// TwinCAT 3 PLC project Untitled1
// ProgramVersion: 3.1.4023.0
// libraries:
//   CmpBitmapPool, * (System)
//   Tc2_Standard, * (Beckhoff Automation GmbH)
//   Tc2_System, * (Beckhoff Automation GmbH)
//   Tc2_Utilities, * (Beckhoff Automation GmbH)
//   Tc3_Module, * (Beckhoff Automation GmbH)
// project tree:
//   / GlobalTextList.TcGTLO, PlcTask.TcTTO, Visualization Manager.TcVMO (not stored)
//   POUs/ MAIN.TcPOU
//   VISUs/ ImagePool.TcIPO (not stored), TextList.TcTLO, Visualization_1.TcVIS, Visualization_2.TcVIS, Visualization_3.TcVIS, VISU_FRAME.TcVIS
// real-time tasks:
//   TASK PlcTask: cycle T#10ms, priority 20, ADS port 350

CONFIGURATION Untitled1
    RESOURCE PLC ON TwinCAT3
        TASK PlcTask(INTERVAL := T#10ms, PRIORITY := 20);
        PROGRAM MAIN WITH PlcTask : MAIN;
    END_RESOURCE
END_CONFIGURATION

// ---- POUs/MAIN.TcPOU
PROGRAM MAIN
VAR
	nState: INT;
	bButton: BOOL;
	ftrig1: F_TRIG;
	bSensor1: BOOL;
	bHat: BOOL;
	rtrig1: R_TRIG;
	bSensor2: BOOL;
	Random1: DRAND;
	nYukseklik: INT;
	sMsgInfo: STRING;
	T1: TON;
	bValf1: BOOL;
	rtrig_Kutu1: R_TRIG;
	rtrig_Kutu2: R_TRIG;
	rtrig_Kutu3: R_TRIG;
	bKutuSensor_1: BOOL;
	bKutuSensor_2: BOOL;
	bKutuSensor_3: BOOL;
	nMalzeme1: INT;
	bValf2: BOOL;
	nMalzeme2: INT;
	bValf3: BOOL;
	nMalzeme3: INT;
	sMsgKisa: STRING(255);
	sMsgOrta: STRING(255);
	sMsgUzun: STRING(255);
	sMsgMalzemeInfo: STRING(255);
	fbSystemTime: FB_LocalSystemTime;
	Year: STRING;
	Month: STRING;
	Day: STRING;
	DMY_LocalTime: STRING;
	HMS_LocalTime: STRING(255);
	Sec: STRING(255);
	Hours: STRING;
	Minute: STRING;
END_VAR



ACT_Uygulama1();
ACT_VisuString();

ACTION ACT_Uygulama1:


ftrig1(CLK:= bSensor1 , Q=> ); // Hattın başında malzeme var mı ?
rtrig1(CLK:= bSensor2 , Q=> ); // Ölçüm yapılacak yerde malzeme var mı ?

rtrig_Kutu1(CLK:= bKutuSensor_1 , Q=> );	// Kısa Boyutlu Malzeme düştü mü kontrolü 
rtrig_Kutu2(CLK:= bKutuSensor_2 , Q=> );	// Orta Boyutlu Malzeme düştü mü kontrolü 
rtrig_Kutu3(CLK:= bKutuSensor_3 , Q=> );	// Uzun Boyutlu Malzeme düştü mü kontrolü 

CASE nState OF
	
	0:
	
		IF bButton THEN 
			
			nState := 10;
			
		END_IF
		
	10:
	
	sMsgInfo := 'Yeni Malzemenin Hatta Aktarılması Bekleniyor';
	
		IF ftrig1.Q THEN
			
			bHat := TRUE;			
			nState := 20;
			
		END_IF
		
	20:
	
	sMsgInfo := 'Malzemenin İstenilen Konuma Gelmesi Bekleniyor';
	
		IF rtrig1.Q THEN
			
			bHat := FALSE;
			
			Random1(Seed:=0 , Num=> );			
			nYukseklik := LREAL_TO_INT((Random1.Num)*100);
			
			nState := 30;
			
		END_IF
	
	30:
	
		IF nYukseklik >= 0 AND nYukseklik <= 30 THEN
			
			nState := 32;
			sMsgInfo := 'Kısa Boyutlu Malzeme.';
		
		ELSIF nYukseklik >30 AND nYukseklik <= 65 THEN

			nState := 34;
			sMsgInfo := 'Orta Boyutlu Malzeme.';

		ELSIF nYukseklik >65 AND nYukseklik <= 100 THEN

			nState := 36;
			sMsgInfo := 'Uzun Boyutlu Malzeme.';
		ELSE 
			sMsgInfo := 'HATA...!';
			nState := 999;
			
		END_IF
		
	32:
	
		bHat := TRUE;
		T1(IN:=TRUE , PT:= T#2S);
		
		IF T1.Q THEN
			nState := 42;
			T1(IN := FALSE);
			bHat := FALSE;
		END_IF
	
	34:
	
		bHat := TRUE;
		T1(IN:=TRUE , PT:= T#4S);
		
		IF T1.Q THEN
			nState := 44;
			T1(IN := FALSE);
			bHat := FALSE;
		END_IF
	
	36:
	
		bHat := TRUE;
		T1(IN:=TRUE , PT:= T#6S);
		
		IF T1.Q THEN
			nState := 46;
			T1(IN := FALSE);
			bHat := FALSE;
		END_IF
		
	42:
	
		bValf1 := TRUE;
		
		sMsgInfo := 'Kısa Boyutlu Malzeme Kutusuna Aktarılıyor.';
		
		IF rtrig_Kutu1.Q THEN
			
			bValf1 := FALSE;
			
			nMalzeme1 := nMalzeme1 + 1; // Kısa boyutlu malzeme sayısını 1 arttır.
			
			nState := 0;
			
		END_IF
		
		
	
	44:
		bValf2 := TRUE;
		
		sMsgInfo := 'Orta Boyutlu Malzeme Kutusuna Aktarılıyor.';
		
		IF rtrig_Kutu2.Q THEN
			
			bValf2 := FALSE;
			
			nMalzeme2 := nMalzeme2 + 1; // Kısa boyutlu malzeme sayısını 1 arttır.
			
			nState := 0;
			
		END_IF
	
	46:
	
		bValf3 := TRUE;
		
		sMsgInfo := 'Uzun Boyutlu Malzeme Kutusuna Aktarılıyor.';
		
		IF rtrig_Kutu3.Q THEN
			
			bValf3 := FALSE;
			
			nMalzeme3 := nMalzeme3 + 1; // Kısa boyutlu malzeme sayısını 1 arttır.
			
			nState := 0;
			
		END_IF
	
		
		
END_CASE

IF NOT bButton THEN
	
	sMsgInfo := 'Sistem Kapalı Durumda.';
	
	nState := 0;
	
	bValf1 := FALSE;
	bValf2 := FALSE;
	bValf3 := FALSE;
	
	bHat := FALSE;
	
	T1(IN:=FALSE);
	
END_IF
END_ACTION

ACTION ACT_VisuString:



sMsgKisa := CONCAT(STR1:='Kısa Boyutlu Malzeme Kutusunda ' , STR2:=INT_TO_STRING(nMalzeme1));
sMsgKisa := CONCAT(STR1:=sMsgKisa , STR2:=' Malzeme Var.' );

sMsgOrta := CONCAT(STR1:='Orta Boyutlu Malzeme Kutusunda ' , STR2:=INT_TO_STRING(nMalzeme2));
sMsgOrta:= CONCAT(STR1:=sMsgOrta , STR2:=' Malzeme Var.' );

sMsgUzun := CONCAT(STR1:='Uzun Boyutlu Malzeme Kutusunda ' , STR2:=INT_TO_STRING(nMalzeme3));
sMsgUzun := CONCAT(STR1:=sMsgUzun , STR2:=' Malzeme Var.' );

sMsgMalzemeInfo := CONCAT(STR1:='Malzeme Boyutu: ' , STR2:=INT_TO_STRING(nYukseklik));
sMsgMalzemeInfo := CONCAT(STR1:=sMsgMalzemeInfo , STR2:='[cm]' );



fbSystemTime(	bEnable:=TRUE );


Year 	:= 	WORD_TO_STRING(fbSystemTime.systemTime.wYear);
Month	:= 	WORD_TO_STRING(fbSystemTime.systemTime.wMonth);
Day 	:= 	WORD_TO_STRING(fbSystemTime.systemTime.wDay);

Hours	:=	WORD_TO_STRING(	fbSystemTime.systemTime.wHour);
Minute	:=  WORD_TO_STRING( fbSystemTime.systemTime.wMinute);
Sec		:=	WORD_TO_STRING( fbSystemTime.systemTime.wSecond);


DMY_LocalTime := CONCAT(STR1:=Day , STR2:='/' );
DMY_LocalTime := CONCAT(STR1:=DMY_LocalTime , STR2:= Month);
DMY_LocalTime := CONCAT(STR1:=DMY_LocalTime , STR2:='/' );
DMY_LocalTime := CONCAT(STR1:=DMY_LocalTime , STR2:=Year );


HMS_LocalTime	:=	CONCAT(STR1:=Hours , STR2:=':' );	
HMS_LocalTime	:=	CONCAT(STR1:=HMS_LocalTime , STR2:=Minute );
HMS_LocalTime	:=	CONCAT(STR1:=HMS_LocalTime , STR2:=':' );	
HMS_LocalTime	:=	CONCAT(STR1:=HMS_LocalTime , STR2:=Sec );
END_ACTION

END_PROGRAM

// ---- GlobalTextList.TcGTLO
TEXTLIST GlobalTextList
  624 = '%s'
  684 = 'Ana Ekran'
  849 = 'Ana Sayfa'
  63 = 'bSensor1'
  479 = 'bSensor2'
  706 = 'Dil Seçeneği'
  637 = 'GroupBox'
  441 = 'Konveyör Hattı'
  907 = 'KutuSensor1'
  970 = 'KutuSensor2'
  179 = 'KutuSensor3'
  389 = 'Sensor Kontrol Bölümü'
  742 = 'Sensor1'
  268 = 'Sensor2'
  823 = 'Sensörler'
  410 = 'Sistem'
  646 = 'Sistem Kontrol'
  207 = 'Türkçe'
  940 = 'Valf1'
  808 = 'Valf2'
  708 = 'Valf3'
  488 = 'Çıkışlar'
  996 = 'İngilizce'
END_TEXTLIST

// ---- VISUs/TextList.TcTLO
TEXTLIST TextList
  0 = 'Sistem' | Türkçe: 'Sistem' | İngilizce: 'System'
  1 = 'Dil Seçeneği' | Türkçe: 'Dil Seçeneği' | İngilizce: 'Languages'
  2 = 'Ana Sayfa' | Türkçe: 'Ana Sayfa' | İngilizce: 'Home Page'
  3 = 'İngilizce' | Türkçe: 'İngilizce' | İngilizce: 'English'
  4 = 'Türkçe' | Türkçe: 'Türkçe' | İngilizce: 'Turkish'
   = ''
END_TEXTLIST

// ---- VISUs/Visualization_1.TcVIS
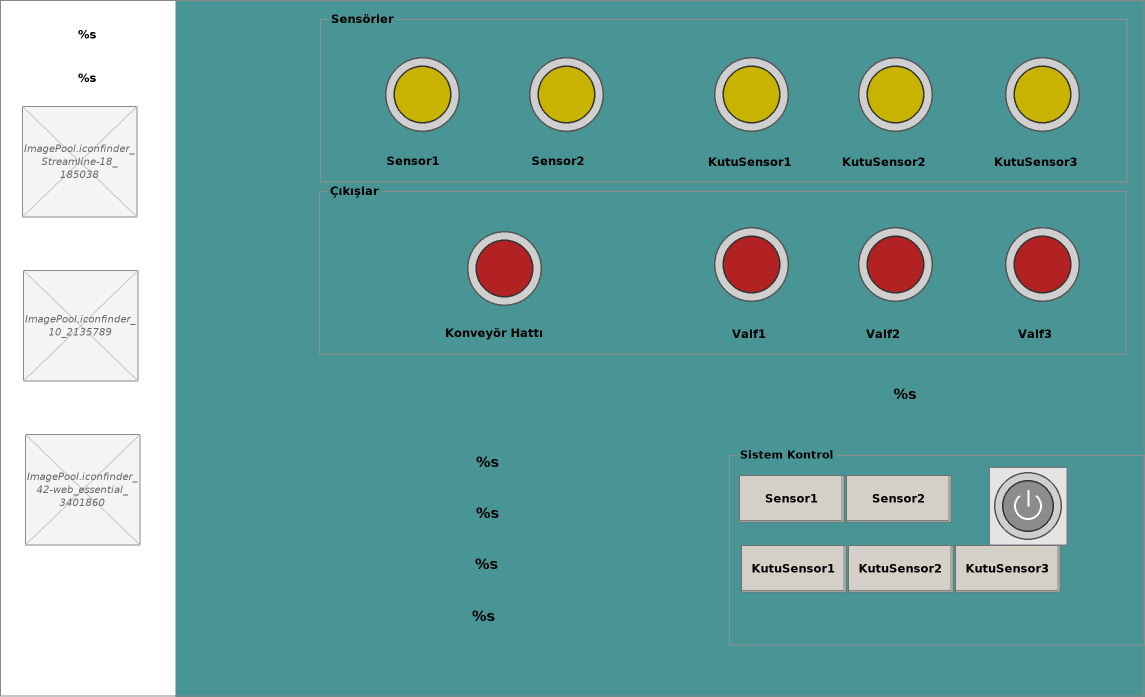
VISUALIZATION Visualization_1  // 1145x697
    Button (739,475 105x47), "Sensor1"
        toggle MAIN.bSensor1
    Button (846,475 105x47), "Sensor2"
        toggle MAIN.bSensor2
    Button (741,545 105x47), "KutuSensor1"
        toggle MAIN.bKutuSensor_1
    Button (848,545 105x47), "KutuSensor2"
        toggle MAIN.bKutuSensor_2
    Button (955,545 105x47), "KutuSensor3"
        toggle MAIN.bKutuSensor_3
    Lamp1 (370,51 105x87), variable: MAIN.bSensor1, style: Lamp-Lamp1-Yellow
    Lamp1 (514,51 105x87), variable: MAIN.bSensor2, style: Lamp-Lamp1-Yellow
    Lamp1 (699,51 105x87), variable: MAIN.bKutuSensor_1, style: Lamp-Lamp1-Yellow
    Lamp1 (843,51 105x87), variable: MAIN.bKutuSensor_2, style: Lamp-Lamp1-Yellow
    Lamp1 (990,51 105x87), variable: MAIN.bKutuSensor_3, style: Lamp-Lamp1-Yellow
    GroupBox (320,11 807x171), "Sensörler"
        Label (42,135 102x30), "Sensor1"
        Label (187,135 102x30), "Sensor2"
        Label (379,136 102x30), "KutuSensor1"
        Label (513,136 102x30), "KutuSensor2"
        Label (665,136 102x30), "KutuSensor3"
    Lamp1 (699,221 105x87), variable: MAIN.bValf1, style: Lamp-Lamp1-Red
    Lamp1 (843,221 105x87), variable: MAIN.bValf2, style: Lamp-Lamp1-Red
    Lamp1 (990,221 105x87), variable: MAIN.bValf3, style: Lamp-Lamp1-Red
    GroupBox (319,183 807x171), "Çıkışlar"
        Label (124,135 102x30), "Konveyör Hattı"
        Label (379,136 102x30), "Valf1"
        Label (513,136 102x30), "Valf2"
        Label (665,136 102x30), "Valf3"
        Lamp1 (133,42 105x87), variable: MAIN.bHat, style: Lamp-Lamp1-Red
    Rectangle (271,440 433x44), "%s", text variable: MAIN.sMsgInfo, text list: ''
    Rectangle (270,491 435x44), "%s", text variable: MAIN.sMsgKisa
    Rectangle (267,542 439x44), "%s", text variable: MAIN.sMsgOrta
    Rectangle (259,594 449x44), "%s", text variable: MAIN.sMsgUzun
    Rectangle (746,372 318x44), "%s", text variable: MAIN.sMsgMalzemeInfo
    Frame (0,0 175x697)
        shows VISU_FRAME(sDayTime := MAIN.DMY_LocalTime, sTime := MAIN.HMS_LocalTime)
    GroupBox (729,447 416x198), "Sistem Kontrol"
        PowerSwitch (257,20 84x78), variable: MAIN.bButton, behaviour: TOGGLE, style: Switch-PowerSwitch-Gray
END_VISUALIZATION

// ---- VISUs/Visualization_2.TcVIS
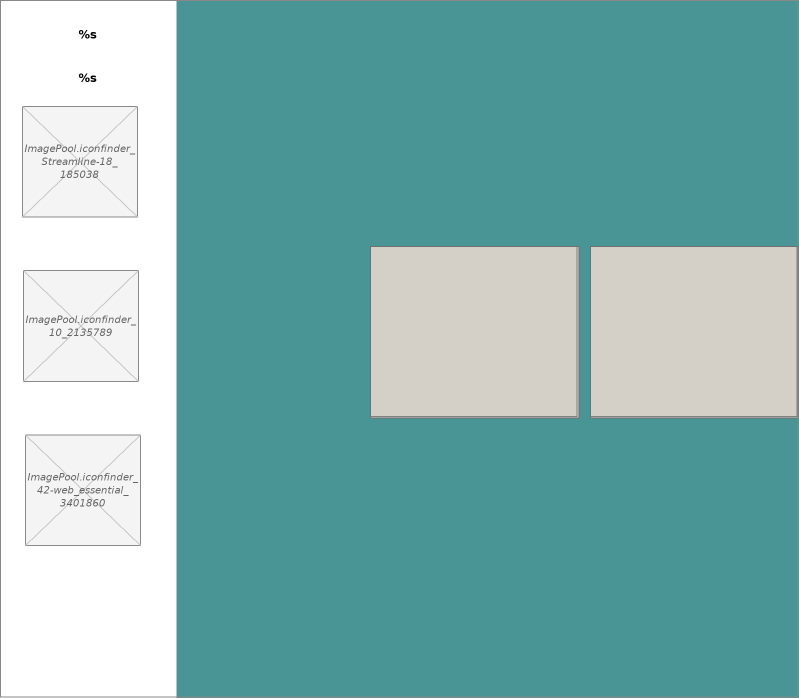
VISUALIZATION Visualization_2  // 799x698
    Button (370,246 209x172), text list: 'TextList', text index: 4
        OnMouseClick: ChangeLanguage ChangeLanguage=Türkçe
    Button (590,246 209x172), text list: 'TextList', text index: 3
        OnMouseClick: ChangeLanguage ChangeLanguage=İngilizce
    Frame (0,0 176x698)
        shows VISU_FRAME(sDayTime := MAIN.DMY_LocalTime, sTime := MAIN.HMS_LocalTime)
END_VISUALIZATION

// ---- VISUs/Visualization_3.TcVIS
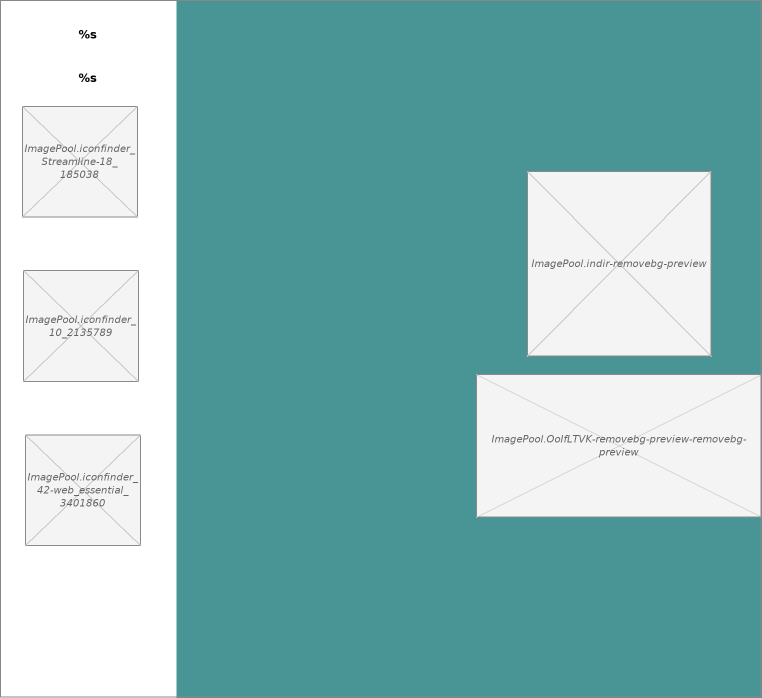
VISUALIZATION Visualization_3  // 762x698
    Image (527,171 184x185), image: ImagePool.indir-removebg-preview
    Image (476,374 286x143), image: ImagePool.OoIfLTVK-removebg-preview-removebg-preview
    Frame (0,0 176x698)
        shows VISU_FRAME(sDayTime := MAIN.DMY_LocalTime, sTime := MAIN.HMS_LocalTime)
END_VISUALIZATION

// ---- VISUs/VISU_FRAME.TcVIS
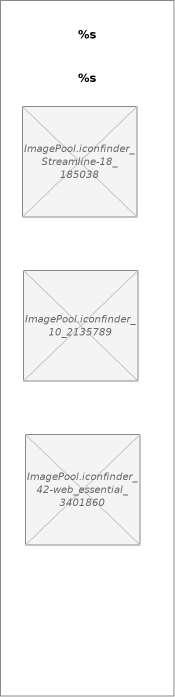
VISUALIZATION VISU_FRAME  // 175x697
VAR_INPUT
	
sDayTime : STRING;
sTime : STRING;

END_VAR
    Rectangle (0,0 175x697)
    Image (23,270 115x111), image: ImagePool.iconfinder_10_2135789
        OnMouseClick: change screen: Visualization_2
    Rectangle (23,385 117x33), text list: 'TextList', text index: 1
    Image (22,106 115x111), image: ImagePool.iconfinder_Streamline-18_185038
        OnMouseClick: change screen: Visualization_3
    Rectangle (22,222 117x33), text list: 'TextList', text index: 2
    Image (25,434 115x111), image: ImagePool.iconfinder_42-web_essential_3401860
        OnMouseClick: change screen: Visualization_1
    Rectangle (25,550 117x33), text list: 'TextList', text index: 0
    Rectangle (12,17 151x35), "%s", text variable: sDayTime
    Rectangle (12,61 151x34), "%s", text variable: sTime
END_VISUALIZATION
